TYPE ST_RoundBeltCoordinates :
STRUCT
	Station : E_RoundBeltStation;
	ReloadCarrier : E_ReloadRoundBelt_PlaceAddress;
END_STRUCT
END_TYPE

(* stored: Version 1.1.0.1, ProductVersion 3.1.4024.13
   DUT ST_RoundBeltCoordinates: Id {11028e02-c3c3-4bac-97eb-34148e547dc9} *)
